PROGRAM MAIN
VAR
END_VAR

END_PROGRAM

(* stored: Version 1.1.0.1
   POU MAIN: Id {a55e4b51-f693-4b56-8bd6-41bb64af543c} *)
